// TIA Portal V19 export
DATA_BLOCK "CEB_2 DB"   // DB135
{ S7_Optimized_Access := 'FALSE' }
   VAR RETAIN
      "DRAIN BY GRAVITY" : Int;
      "CEB BACKWASH_1" : Int;
      "CEB BACKWASH_2" : Int;
      SOAK : Int;
      BACKWASH_1 : Int;
      BACKWASH_2 : Int;
      "DRAIN BY GRAVITY_2" : Int;
      "TOTAL CYCLE" : Int;
      PV : Struct
         "DRAIN BY GRAVITY" : Int;
         "CEB BACKWASH_1" : Int;
         "CEB BACKWASH_2" : Int;
         SOAK : Int;
         BACKWASH_1 : Int;
         BACKWASH_2 : Int;
         "DRAIN BY GRAVITY_2" : Int;
         "TOTAL CYCLE" : Int;
      END_STRUCT;
   END_VAR
BEGIN
END_DATA_BLOCK
